TYPE udt_EL6900_SafetyGroup_CMD :
	STRUCT
	Run_Stop: BOOL;
	Error_Ack: BOOL;
	FB_Restart: ARRAY[0..31] OF BOOL;
	END_STRUCT
END_TYPE

(* stored: Version 1.1.0.1, ProductVersion 3.1.4024.9
   DUT udt_EL6900_SafetyGroup_CMD: Id {d49e1a1e-2a6f-4655-a7c4-59e8e2c308a8} *)
